// TwinCAT 3 PLC project ComissioningPlc
// ProgramVersion: 3.1.4026.24
// libraries:
//   Tc2_MC2, * (Beckhoff Automation GmbH)
//   Tc2_Standard, * (Beckhoff Automation GmbH)
//   Tc2_System, * (Beckhoff Automation GmbH)
//   Tc3_LmDualAxisCoordinator, * (Milan Lazov)
// project tree:
//   DUTs/STRUCTs/Physical/ ST_Axis_Physical_In.TcDUT, ST_Axis_Physical_Out.TcDUT
//   DUTs/STRUCTs/Public %28Interface%29/ ST_AxisHmiCmd.TcDUT (not stored), ST_AxisHmiStatus.TcDUT (not stored), ST_AxisInterface.TcDUT (not stored), ST_DualDriveInterface.TcDUT (not stored)
//   GVLs/ GVL_IO.TcGVL, GVL_Motion.TcGVL
//   / PlcTask.TcTTO
//   POUs/ FB_AxisInputMapping.TcPOU, FB_AxisOutputMapping.TcPOU, MAIN.TcPOU
// real-time tasks:
//   TASK PlcTask: cycle T#10ms, priority 20, ADS port 350
// motion (NC):
//   TASK NC-Task 1 SAF: cycle T#2ms, priority 4, ADS port 501
//   TASK NC-Task 1 SVB: cycle T#10ms, priority 8, ADS port 511
//   AXIS Axis_M (id 1)
//     OtherSettings: AllowMotionCmdToSlave=true
//     encoder EncType=19
//       EncPara: MaxCount=#xffffffff
//     drive DrvType=16
//       DrvPara: MaxCount=#xffffffff, DriveControlDWord=#x00020100
//         Analog: TorqueSetpointScale=10, ScaleFactorActTorque=0.1
//         TimeComp: TaskDelayCycles=1
//     controller CtrType=1
//       CtrPara: PriorControlFactor=1
//         Observer: BandWidth=20
//   AXIS Axis_S (id 2)
//     OtherSettings: AllowMotionCmdToSlave=true
//     encoder EncType=19
//       EncPara: MaxCount=#xffffffff
//     drive DrvType=16
//       DrvPara: MaxCount=#xffffffff, DriveControlDWord=#x00020100
//         Analog: TorqueSetpointScale=10, ScaleFactorActTorque=0.1
//         TimeComp: TaskDelayCycles=1
//     controller CtrType=1
//       CtrPara: PriorControlFactor=1
//         Observer: BandWidth=20
// I/O:
//   DEVICE Device 1 (EtherCAT) (disabled), AmsNetId 192.168.0.14.2.1
//     Master (i950 (BS-STO)) [i950 (BS-STO) FW V01.14 - TA CiA402 Advanced (1) V00]
//       modules: Module 1 (Universal (CSP + Speed and Torque Limits))
//     Slave (i950 (BS-STO)) [i950 (BS-STO) FW V01.14 - TA CiA402 Advanced (1) V00]
//       modules: Module 1 (Universal (CSP + Speed and Torque Limits))
//     Coupler (EK1100) [EK1100 EtherCAT Coupler (2A E-Bus)]
//       Master (EL1809) [EL1809 16Ch. Dig. Input 24V, 3ms]
//       Slave (EL1809) [EL1809 16Ch. Dig. Input 24V, 3ms]
// variable links:
//   NC-Task 1 SAF/Axes/Axis_M <-> Device 1 (EtherCAT)/Master (i950 (BS-STO))
//     Drive/Inputs/In/nDataIn1 <-> Module 1 (Universal (CSP + Speed and Torque Limits))/Inputs/Following error actual value
//     Drive/Inputs/In/nDataIn3[0] <-> Module 1 (Universal (CSP + Speed and Torque Limits))/Inputs/Actual torque
//     Drive/Inputs/In/nState1 <-> Module 1 (Universal (CSP + Speed and Torque Limits))/Inputs/CiA status word
//     Drive/Inputs/In/nState2 <-> Module 1 (Universal (CSP + Speed and Torque Limits))/Inputs/CiA status word @bit 8
//     Drive/Inputs/In/nState4 @bit 1 <-> WcState/InputToggle
//     Drive/Inputs/In/nState4 <-> WcState/WcState
//     Drive/Inputs/In/nState5 <-> Module 1 (Universal (CSP + Speed and Torque Limits))/Inputs/CiA: Active operation mode
//     Drive/Outputs/Out/nCtrl1 <-> Module 1 (Universal (CSP + Speed and Torque Limits))/Outputs/CiA control word
//     Drive/Outputs/Out/nCtrl2 <-> Module 1 (Universal (CSP + Speed and Torque Limits))/Outputs/CiA control word @bit 8
//     Drive/Outputs/Out/nCtrl5 <-> Module 1 (Universal (CSP + Speed and Torque Limits))/Outputs/CiA: Operation mode
//     Drive/Outputs/Out/nDataOut1 <-> Module 1 (Universal (CSP + Speed and Torque Limits))/Outputs/Set position
//     Drive/Outputs/Out/nDataOut3[0] <-> Module 1 (Universal (CSP + Speed and Torque Limits))/Outputs/Offset torque
//     Enc/Inputs/In/nDataIn1 <-> Module 1 (Universal (CSP + Speed and Torque Limits))/Inputs/Actual position
//     Enc/Inputs/In/nDataIn3 <-> Module 1 (Universal (CSP + Speed and Torque Limits))/Touchprobe Inputs/Touch probe 1: Position at pos. edge
//     Enc/Inputs/In/nDataIn5 <-> Module 1 (Universal (CSP + Speed and Torque Limits))/Touchprobe Inputs/Touch probe 2: Position at pos. edge
//     Enc/Inputs/In/nDataIn4 <-> Module 1 (Universal (CSP + Speed and Torque Limits))/Touchprobe Inputs/Touch probe 1: Position at neg. edge
//     Enc/Inputs/In/nDataIn6 <-> Module 1 (Universal (CSP + Speed and Torque Limits))/Touchprobe Inputs/Touch probe 2: Position at neg. edge
//     Enc/Inputs/In/nDataIn7 <-> Module 1 (Universal (CSP + Speed and Torque Limits))/Inputs/Actual speed
//     Enc/Inputs/In/nState4 @bit 1 <-> WcState/InputToggle
//     Enc/Inputs/In/nState4 <-> WcState/WcState
//     Enc/Inputs/In/nState5 <-> Module 1 (Universal (CSP + Speed and Torque Limits))/Touchprobe Inputs/Touch probe status
//     Enc/Inputs/In/nState6 <-> Module 1 (Universal (CSP + Speed and Torque Limits))/Touchprobe Inputs/Touch probe status @bit 8
//     Enc/Outputs/Out/nCtrl5 <-> Module 1 (Universal (CSP + Speed and Torque Limits))/Touchprobe Outputs/Touch probe settings
//     Enc/Outputs/Out/nCtrl6 <-> Module 1 (Universal (CSP + Speed and Torque Limits))/Touchprobe Outputs/Touch probe settings @bit 8
//   NC-Task 1 SAF/Axes/Axis_S <-> Device 1 (EtherCAT)/Slave (i950 (BS-STO))
//     Drive/Inputs/In/nDataIn1 <-> Module 1 (Universal (CSP + Speed and Torque Limits))/Inputs/Following error actual value
//     Drive/Inputs/In/nDataIn3[0] <-> Module 1 (Universal (CSP + Speed and Torque Limits))/Inputs/Actual torque
//     Drive/Inputs/In/nState1 <-> Module 1 (Universal (CSP + Speed and Torque Limits))/Inputs/CiA status word
//     Drive/Inputs/In/nState2 <-> Module 1 (Universal (CSP + Speed and Torque Limits))/Inputs/CiA status word @bit 8
//     Drive/Inputs/In/nState4 @bit 1 <-> WcState/InputToggle
//     Drive/Inputs/In/nState4 <-> WcState/WcState
//     Drive/Inputs/In/nState5 <-> Module 1 (Universal (CSP + Speed and Torque Limits))/Inputs/CiA: Active operation mode
//     Drive/Outputs/Out/nCtrl1 <-> Module 1 (Universal (CSP + Speed and Torque Limits))/Outputs/CiA control word
//     Drive/Outputs/Out/nCtrl2 <-> Module 1 (Universal (CSP + Speed and Torque Limits))/Outputs/CiA control word @bit 8
//     Drive/Outputs/Out/nCtrl5 <-> Module 1 (Universal (CSP + Speed and Torque Limits))/Outputs/CiA: Operation mode
//     Drive/Outputs/Out/nDataOut1 <-> Module 1 (Universal (CSP + Speed and Torque Limits))/Outputs/Set position
//     Drive/Outputs/Out/nDataOut3[0] <-> Module 1 (Universal (CSP + Speed and Torque Limits))/Outputs/Offset torque
//     Enc/Inputs/In/nDataIn1 <-> Module 1 (Universal (CSP + Speed and Torque Limits))/Inputs/Actual position
//     Enc/Inputs/In/nDataIn3 <-> Module 1 (Universal (CSP + Speed and Torque Limits))/Touchprobe Inputs/Touch probe 1: Position at pos. edge
//     Enc/Inputs/In/nDataIn5 <-> Module 1 (Universal (CSP + Speed and Torque Limits))/Touchprobe Inputs/Touch probe 2: Position at pos. edge
//     Enc/Inputs/In/nDataIn4 <-> Module 1 (Universal (CSP + Speed and Torque Limits))/Touchprobe Inputs/Touch probe 1: Position at neg. edge
//     Enc/Inputs/In/nDataIn6 <-> Module 1 (Universal (CSP + Speed and Torque Limits))/Touchprobe Inputs/Touch probe 2: Position at neg. edge
//     Enc/Inputs/In/nDataIn7 <-> Module 1 (Universal (CSP + Speed and Torque Limits))/Inputs/Actual speed
//     Enc/Inputs/In/nState4 @bit 1 <-> WcState/InputToggle
//     Enc/Inputs/In/nState4 <-> WcState/WcState
//     Enc/Inputs/In/nState5 <-> Module 1 (Universal (CSP + Speed and Torque Limits))/Touchprobe Inputs/Touch probe status
//     Enc/Inputs/In/nState6 <-> Module 1 (Universal (CSP + Speed and Torque Limits))/Touchprobe Inputs/Touch probe status @bit 8
//     Enc/Outputs/Out/nCtrl5 <-> Module 1 (Universal (CSP + Speed and Torque Limits))/Touchprobe Outputs/Touch probe settings
//     Enc/Outputs/Out/nCtrl6 <-> Module 1 (Universal (CSP + Speed and Torque Limits))/Touchprobe Outputs/Touch probe settings @bit 8
//   ComissioningPlc/ComissioningPlc Instance <-> Device 1 (EtherCAT)/Coupler (EK1100)/Master (EL1809)
//     PlcTask Inputs/GVL_IO.stMaster_Physical_In/xCalibrationCam <-> Channel 11/Input
//     PlcTask Inputs/GVL_IO.stMaster_Physical_In/xHaltBtn <-> Channel 8/Input
//     PlcTask Inputs/GVL_IO.stMaster_Physical_In/xHomeBtn <-> Channel 10/Input
//     PlcTask Inputs/GVL_IO.stMaster_Physical_In/xJogBkwFastBtn <-> Channel 4/Input
//     PlcTask Inputs/GVL_IO.stMaster_Physical_In/xJogBkwSlowBtn <-> Channel 5/Input
//     PlcTask Inputs/GVL_IO.stMaster_Physical_In/xJogFwdFastBtn <-> Channel 7/Input
//     PlcTask Inputs/GVL_IO.stMaster_Physical_In/xJogFwdSlowBtn <-> Channel 6/Input
//     PlcTask Inputs/GVL_IO.stMaster_Physical_In/xMoveAbsBtn <-> Channel 2/Input
//     PlcTask Inputs/GVL_IO.stMaster_Physical_In/xMoveVeloBtn <-> Channel 3/Input
//     PlcTask Inputs/GVL_IO.stMaster_Physical_In/xPowerEnableBtn <-> Channel 1/Input
//     PlcTask Inputs/GVL_IO.stMaster_Physical_In/xResetBtn <-> Channel 12/Input
//     PlcTask Inputs/GVL_IO.stMaster_Physical_In/xStopBtn <-> Channel 9/Input
//   ComissioningPlc/ComissioningPlc Instance <-> Device 1 (EtherCAT)/Coupler (EK1100)/Slave (EL1809)
//     PlcTask Inputs/GVL_IO.stSlave_Physical_In/xCalibrationCam <-> Channel 11/Input
//     PlcTask Inputs/GVL_IO.stSlave_Physical_In/xHaltBtn <-> Channel 8/Input
//     PlcTask Inputs/GVL_IO.stSlave_Physical_In/xHomeBtn <-> Channel 10/Input
//     PlcTask Inputs/GVL_IO.stSlave_Physical_In/xJogBkwFastBtn <-> Channel 4/Input
//     PlcTask Inputs/GVL_IO.stSlave_Physical_In/xJogBkwSlowBtn <-> Channel 5/Input
//     PlcTask Inputs/GVL_IO.stSlave_Physical_In/xJogFwdFastBtn <-> Channel 7/Input
//     PlcTask Inputs/GVL_IO.stSlave_Physical_In/xJogFwdSlowBtn <-> Channel 6/Input
//     PlcTask Inputs/GVL_IO.stSlave_Physical_In/xMoveAbsBtn <-> Channel 2/Input
//     PlcTask Inputs/GVL_IO.stSlave_Physical_In/xMoveVeloBtn <-> Channel 3/Input
//     PlcTask Inputs/GVL_IO.stSlave_Physical_In/xPowerEnableBtn <-> Channel 1/Input
//     PlcTask Inputs/GVL_IO.stSlave_Physical_In/xResetBtn <-> Channel 12/Input
//     PlcTask Inputs/GVL_IO.stSlave_Physical_In/xStopBtn <-> Channel 9/Input
//   ComissioningPlc/ComissioningPlc Instance <-> NC-Task 1 SAF/Axes/Axis_M
//     PlcTask Inputs/GVL_Motion.Axis_M.NcToPlc <-> Outputs/ToPlc
//     PlcTask Outputs/GVL_Motion.Axis_M.PlcToNc <-> Inputs/FromPlc
//   ComissioningPlc/ComissioningPlc Instance <-> NC-Task 1 SAF/Axes/Axis_S
//     PlcTask Inputs/GVL_Motion.Axis_S.NcToPlc <-> Outputs/ToPlc
//     PlcTask Outputs/GVL_Motion.Axis_S.PlcToNc <-> Inputs/FromPlc

CONFIGURATION ComissioningPlc
    RESOURCE PLC ON TwinCAT3
        TASK PlcTask(INTERVAL := T#10ms, PRIORITY := 20);
        PROGRAM MAIN WITH PlcTask : MAIN;
    END_RESOURCE
END_CONFIGURATION

// ---- DUTs/STRUCTs/Physical/ST_Axis_Physical_In.TcDUT
// ==============================================================================
// DUT:            ST_Axis_Physical_In
// Description:    Hardware digital input signals from operator buttons and panel switches.
// ==============================================================================
TYPE ST_Axis_Physical_In :
STRUCT
    // --- Drive Power Stage ---
    xPowerEnableBtn   : BOOL; /// Drive power enable button (Normally Open)

    // --- Autonomous Motion Initiation ---
    xMoveAbsBtn       : BOOL; /// Absolute move start button (Normally Open)
    xMoveVeloBtn      : BOOL; /// Velocity move start button (Normally Open)

    // --- Manual Continuous Jogging ---
    xJogBkwFastBtn    : BOOL; /// Fast reverse manual jog button (Normally Open)
    xJogBkwSlowBtn    : BOOL; /// Slow reverse manual jog button (Normally Open)
    xJogFwdSlowBtn    : BOOL; /// Slow forward manual jog button (Normally Open)
    xJogFwdFastBtn    : BOOL; /// Fast forward manual jog button (Normally Open)

    // --- Standstill, Calibration & Diagnostics ---
    xHaltBtn          : BOOL; /// Controlled deceleration halt button (Normally Open)
    xStopBtn          : BOOL; /// Hardware stop button (Normally Open)
    xHomeBtn          : BOOL; /// Reference homing start button (Normally Open)
	xCalibrationCam   : BOOL; /// Reference homing calibration cam or proximity sensor (Normally Open)
    xResetBtn         : BOOL; /// Fault reset acknowledgment button (Normally Open)
END_STRUCT
END_TYPE

// ---- DUTs/STRUCTs/Physical/ST_Axis_Physical_Out.TcDUT
// ==============================================================================
// DUT:            ST_Axis_Physical_In
// Description:    Hardware digital output signals driving panel indicators, pilot lamps, or field actuators.
// ==============================================================================
TYPE ST_Axis_Physical_Out :
STRUCT
    // Reserved for field hardware outputs (e.g., status pilot lamps, mechanical brake coils)
END_STRUCT
END_TYPE

// ---- GVLs/GVL_IO.TcGVL
// ==============================================================================
// GVL:            GVL_IO
// Description:    Global variable list mapping physical fieldbus process inputs 
//                 from digital terminal slices (%I*) for master and slave axes.
// ==============================================================================
{attribute 'qualified_only'}
VAR_GLOBAL
    // Hardware digital input images linked to terminal slice channels (%I*)
    stMaster_Physical_In AT %I* : ST_Axis_Physical_In; // Master axis physical pushbuttons and panel switches
    stSlave_Physical_In  AT %I* : ST_Axis_Physical_In; // Slave axis physical pushbuttons and panel switches
END_VAR

// ---- GVLs/GVL_Motion.TcGVL
// ==============================================================================
// GVL:            GVL_Motion
// Description:    Global variable list instantiating TwinCAT NC axis hardware 
//                 references (AXIS_REF) and composite HMI visualization nodes.
// ==============================================================================
{attribute 'qualified_only'}
VAR_GLOBAL
    // --- Master Motion Axis ---
    Axis_M               : AXIS_REF;               // TwinCAT NC axis reference for Master axis
    Axis_M_Interface     : ST_AxisInterface;       // Visualization interface node for Master axis
    
    // --- Slave Motion Axis ---
    Axis_S               : AXIS_REF;               // TwinCAT NC axis reference for Slave axis
    Axis_S_Interface     : ST_AxisInterface;       // Visualization interface node for Slave axis

    // --- Dual-Drive Coordination Module ---
    DualDrive_Interface  : ST_DualDriveInterface;  // Visualization interface node for Dual-Drive equipment module
END_VAR

// ---- POUs/MAIN.TcPOU
// ==============================================================================
// POU:            MAIN
// Description:    Top-level application program coordinating ingress signal mapping, 
//                 dual-drive motion control execution, and HMI telemetry egress.
// ==============================================================================
PROGRAM MAIN
VAR
    // --- Application Mapping & Execution Instances ---
    fbMasterAxisInputMapping  : FB_AxisInputMapping;  // Combines HMI and physical panel inputs for Master axis
    fbSlaveAxisInputMapping   : FB_AxisInputMapping;  // Combines HMI and physical panel inputs for Slave axis
    
    fbAxisDualDrive           : FB_AxisDualDrive;     // Core dual-axis equipment module coordinating motion & gearing
    
    fbMasterAxisOutputMapping : FB_AxisOutputMapping; // Packs Master telemetry and diagnostics for HMI display
    fbSlaveAxisOutputMapping  : FB_AxisOutputMapping; // Packs Slave telemetry and diagnostics for HMI display

    // --- Master Axis Local Process Data ---
    stMasterAxisSystemCmd     : ST_AxisSystemCmd;     // Arbitrated command pipeline dispatched to Master axis
    stMasterFeedback          : ST_AxisFeedback;      // Live cyclic NC feedback image for Master axis
    eMasterState              : E_AxisState;          // Active operational state of Master axis controller
    udiMasterErrorId          : UDINT;                // Active diagnostic error code for Master axis

    // --- Slave Axis Local Process Data ---
    stSlaveAxisSystemCmd      : ST_AxisSystemCmd;     // Arbitrated command pipeline dispatched to Slave axis
    stSlaveFeedback           : ST_AxisFeedback;      // Live cyclic NC feedback image for Slave axis
    eSlaveState               : E_AxisState;          // Active operational state of Slave axis controller
    udiSlaveErrorId           : UDINT;                // Active diagnostic error code for Slave axis
END_VAR

// 1. Ingress Command Mapping: Condition HMI and physical buttons for Master axis
fbMasterAxisInputMapping(
    stHmiCmd     := GVL_Motion.Axis_M_Interface.stHmiCmd,
    stPhysicalIn := GVL_IO.stMaster_Physical_In,
	
    stSystemCmd  => stMasterAxisSystemCmd
);

// 2. Ingress Command Mapping: Condition HMI and physical buttons for Slave axis
fbSlaveAxisInputMapping(
    stHmiCmd     := GVL_Motion.Axis_S_Interface.stHmiCmd,
    stPhysicalIn := GVL_IO.stSlave_Physical_In,
	
    stSystemCmd  => stSlaveAxisSystemCmd
);

// 3. Dual-Drive Coordination: Execute master-slave gearing, power policies, and motion
fbAxisDualDrive(
    eCouplingPolicy       := GVL_Motion.DualDrive_Interface.eCouplingPolicy,
    eDriveType            := GVL_Motion.DualDrive_Interface.eDriveType,
    lrRatioNumerator      := GVL_Motion.DualDrive_Interface.lrRatioNumerator,
    iRatioDenominator     := GVL_Motion.DualDrive_Interface.iRatioDenominator,
    xCmdGearIn            := GVL_Motion.DualDrive_Interface.xCmdGearIn,
    xCmdGearOut           := GVL_Motion.DualDrive_Interface.xCmdGearOut,
    xCmdReset             := GVL_Motion.DualDrive_Interface.xCmdReset,
    xMasterCalibrationCam := GVL_IO.stMaster_Physical_In.xCalibrationCam,
    xSlaveCalibrationCam  := GVL_IO.stSlave_Physical_In.xCalibrationCam,
	
    Axis_Master           := GVL_Motion.Axis_M,
    Axis_M_Cmd            := stMasterAxisSystemCmd,
    Axis_M_Config         := GVL_Motion.Axis_M_Interface.stConfig,
    
    Axis_Slave            := GVL_Motion.Axis_S,
    Axis_S_Cmd            := stSlaveAxisSystemCmd,
    Axis_S_Config         := GVL_Motion.Axis_S_Interface.stConfig,
    
    eAxisCouplingState    => GVL_Motion.DualDrive_Interface.eAxisCouplingState,
	xRegearRequired       => GVL_Motion.DualDrive_Interface.xRegearRequired,
	lrActiveRatioNum      => GVL_Motion.DualDrive_Interface.lrActiveRatioNum,
    uiActiveRatioDenom    => GVL_Motion.DualDrive_Interface.uiActiveRatioDenom,
    xError                => GVL_Motion.DualDrive_Interface.xError,
    udiErrorId            => GVL_Motion.DualDrive_Interface.udiErrorId,
    
    eMasterState          => eMasterState,
    udiMasterErrorId      => udiMasterErrorId,
    eSlaveState           => eSlaveState,
    udiSlaveErrorId       => udiSlaveErrorId,
    stMasterFeedback      => stMasterFeedback,
    stSlaveFeedback       => stSlaveFeedback
);

// 4. Egress Telemetry Mapping: Pack Master states and diagnostics for visualization
fbMasterAxisOutputMapping(
    eCurrentState := eMasterState,
    udiErrorId    := udiMasterErrorId,
    stFeedback    := stMasterFeedback,
    stHmiStatus   => GVL_Motion.Axis_M_Interface.stHmiStatus
);

// 5. Egress Telemetry Mapping: Pack Slave states and diagnostics for visualization
fbSlaveAxisOutputMapping(
    eCurrentState := eSlaveState,
    udiErrorId    := udiSlaveErrorId,
    stFeedback    := stSlaveFeedback,
    stHmiStatus   => GVL_Motion.Axis_S_Interface.stHmiStatus
);

END_PROGRAM

// ---- POUs/FB_AxisInputMapping.TcPOU
// ==============================================================================
// POU:            FB_AxisInputMapping
// Description:    Commissioning & VISU helper block. Combines parallel HMI 
//                 visualization commands and physical panel pushbuttons into 
//                 a unified ST_AxisSystemCmd structure for axis controllers.
// ==============================================================================
FUNCTION_BLOCK FB_AxisInputMapping
VAR_IN_OUT CONSTANT
    // Read-only reference to asynchronous commands coming from the HMI screen
    stHmiCmd      : ST_AxisHmiCmd;

    // Read-only reference to hardwired pushbuttons and physical panel inputs
    stPhysicalIn  : ST_Axis_Physical_In;
END_VAR

VAR_OUTPUT
    // Conditioned internal command structure dispatched to FB_AxisController or FB_AxisDualDrive
    stSystemCmd   : ST_AxisSystemCmd;
END_VAR

VAR
    // Edge-conditioning instances to generate single-cycle execution pulses from HMI/panel signals
    fbCmdMoveAbs  : FB_InputEdgeDetection; // Filters absolute move requests into a 1-cycle pulse
    fbCmdMoveVelo : FB_InputEdgeDetection; // Filters velocity move requests into a 1-cycle pulse
    fbCmdHalt     : FB_InputEdgeDetection; // Filters halt requests into a 1-cycle pulse
    fbCmdHome     : FB_InputEdgeDetection; // Filters homing calibration requests into a 1-cycle pulse
    fbCmdReset    : FB_InputEdgeDetection; // Filters error reset requests into a 1-cycle pulse
END_VAR

// ==============================================================================
// 1. PULSED MOTION COMMAND CONDITIONING (EDGE-TRIGGERED)
// ==============================================================================
// Evaluates HMI and physical pushbuttons in parallel. Passes signals through
// FB_InputEdgeDetection instances to ensure that sustained presses or latched
// buttons produce exactly one execution pulse on the outgoing command pipeline.

// Absolute Positioning Command
fbCmdMoveAbs(
    xHmiInput      := stHmiCmd.xMoveAbs,
    xPhysicalInput := stPhysicalIn.xMoveAbsBtn
);  
stSystemCmd.xMoveAbs := fbCmdMoveAbs.xPulsedCmd;

// Continuous Velocity Command
fbCmdMoveVelo(
    xHmiInput      := stHmiCmd.xMoveVelo,
    xPhysicalInput := stPhysicalIn.xMoveVeloBtn
);  
stSystemCmd.xMoveVelo := fbCmdMoveVelo.xPulsedCmd;

// Controlled Halt Command
fbCmdHalt(
    xHmiInput      := stHmiCmd.xHalt,
    xPhysicalInput := stPhysicalIn.xHaltBtn
);  
stSystemCmd.xHalt := fbCmdHalt.xPulsedCmd;

// Axis Calibration / Homing Command
fbCmdHome(
    xHmiInput      := stHmiCmd.xHome,
    xPhysicalInput := stPhysicalIn.xHomeBtn
);  
stSystemCmd.xHome := fbCmdHome.xPulsedCmd;

// Fault Reset Command
fbCmdReset(
    xHmiInput      := stHmiCmd.xReset,
    xPhysicalInput := stPhysicalIn.xResetBtn
);  
stSystemCmd.xReset := fbCmdReset.xPulsedCmd;

// ==============================================================================
// 2. CONTINUOUS & INTERLOCK COMMAND MAPPING (LEVEL-TRIGGERED)
// ==============================================================================
// Evaluated directly without edge detection. These signals represent operational 
// states or sustained operator holds that must persist across scan cycles.

// Operational Stop (Asserted as long as either HMI stop or physical stop button is active)
stSystemCmd.xStop        := stHmiCmd.xStop OR stPhysicalIn.xStopBtn;

// Software Power Enable (Direct mapping from HMI enable toggle or physical enable button)
stSystemCmd.xPowerEnable := stHmiCmd.xPowerEnable OR stPhysicalIn.xPowerEnableBtn;

// Manual Jogging Vectors (Active while operator maintains button press)
stSystemCmd.xJogBkwFast  := stHmiCmd.xJogBkwFast OR stPhysicalIn.xJogBkwFastBtn;
stSystemCmd.xJogBkwSlow  := stHmiCmd.xJogBkwSlow OR stPhysicalIn.xJogBkwSlowBtn;
stSystemCmd.xJogFwdSlow  := stHmiCmd.xJogFwdSlow OR stPhysicalIn.xJogFwdSlowBtn;
stSystemCmd.xJogFwdFast  := stHmiCmd.xJogFwdFast OR stPhysicalIn.xJogFwdFastBtn;

END_FUNCTION_BLOCK

// ---- POUs/FB_AxisOutputMapping.TcPOU
// ==============================================================================
// POU:            FB_AxisOutputMapping
// Description:    Commissioning & VISU helper block. Packs live axis controller
//                 states, diagnostic fault codes, and cyclic NC feedback into 
//                 the ST_AxisHmiStatus structure for visualization displays.
// ==============================================================================
FUNCTION_BLOCK FB_AxisOutputMapping
VAR_INPUT
    // Operational state machine state reported by FB_AxisController or FB_AxisDualDrive
    eCurrentState : E_AxisState;

    // Active diagnostic error ID reported by the controller
    udiErrorId    : UDINT;
END_VAR

VAR_IN_OUT CONSTANT
    // Read-only reference to the live NC feedback image (position, velocity, status flags)
    stFeedback    : ST_AxisFeedback;
END_VAR

VAR_OUTPUT
    // Consolidated status structure bound to HMI visualization elements and indicators
    stHmiStatus   : ST_AxisHmiStatus;
END_VAR

// ==============================================================================
// 1. VISUALIZATION STATUS AGGREGATION & MAPPING
// ==============================================================================
// Combines low-level NC cyclic telemetry with high-level controller states 
// and diagnostic fault codes into a single structure for direct VISU/HMI binding.

// Discrete Status Flags
stHmiStatus.xPowerActive  := stFeedback.xPowerActive;
stHmiStatus.xReady        := stFeedback.xReady;
stHmiStatus.xMoving       := stFeedback.xMoving;
stHmiStatus.xInPosition   := stFeedback.xInPosition;
stHmiStatus.xError        := (eCurrentState = E_AxisState.ERROR);

// Diagnostic Telemetry & State Machine Tracking
stHmiStatus.udiErrorId    := udiErrorId;
stHmiStatus.eCurrentState := eCurrentState;
stHmiStatus.xInGear 	  := stFeedback.xInGear;

// Live Kinematic Process Data
stHmiStatus.lrActPos      := stFeedback.lrActPos;
stHmiStatus.lrActVel      := stFeedback.lrActVel;

END_FUNCTION_BLOCK
